# EPICS StreamDevice protocol: gardasoftLED/RTSeries.protocol
# Protocol file for the Gardasoft Vision RT series LED lighting controllers (tested on the RT460-20)
# Version: 1.0
# Date:    14-02-2011

# Please refer to the Gardasoft Vision User Manual Revision 3
# Comms settings: 115200,8,N,1

OutTerminator = CR;
InTerminator = LF CR ">";
replytimeout = 100;
readtimeout  = 2000;

# Report the firmware version
getVersion {
	out "VR";
	in "VR%(\$1:MODEL)s %(\$1:HW_VERSION)s %(\$1:FW_VERSION)s";
}

# Save settings to the controller's
# non-volatile memory
save {
	out "AW";
	in "AW";
}

# Clear errors.  The errors that were cleared
# are saved as a String
resetErrors {
	out "GR";
	in "%s";
}

# Set the max current rating for a light (mA)
# $1 - output channel
# $2 - PV prefix
setRating {
	out "VL\$1,0,%fma";
	in "VL\$1,%(\$2:MAXVOLTAGE)f,%(\$2:MAXCURRENT)fMA";
}

# Set the max voltage rating for a light (V)
# $1 - output channel
# $2 - PV prefix
setVoltageRating {
	out "VL\$1,%f,0";
	in "VL\$1,%(\$2:MAXVOLTAGE)f,%(\$2:MAXCURRENT)f";
}

# Set continuous output (at a percentage of full brightness)
# $1 - output channel
# $2 - PV prefix
setOutput {
	out "RS\$1,%u";
	in "RS\$1,%(\$2:BRIGHTNESS)f";
}

# Set the option flags (at a percentage of full brightness)
# $1 - output channel
# $2 - PV prefix
setOptionFlags {
	out "RE\$1,%u";
	in "RE\$1,%(\$2:OPTIONS)f";
}
